RoboDK station: RDTSDemoBasketLineAndAGV.rdk

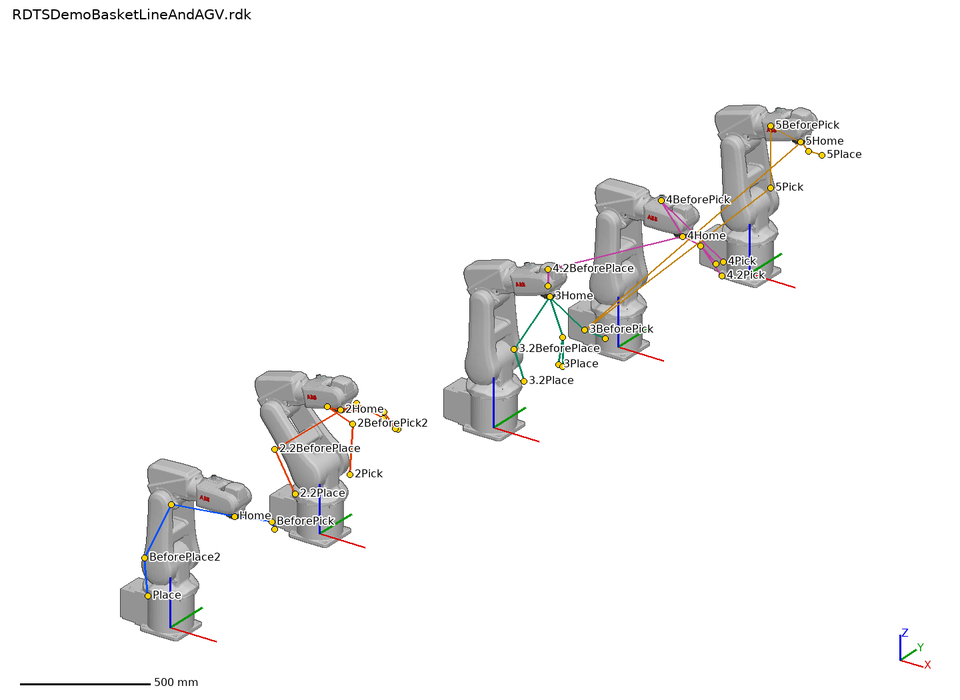
[picture v0: the station drawn from its stored meshes, robots at their saved joint values, targets as dots, program paths as lines]
Station RDTSDemoBasketLine (saved by RoboDK 5.6.0). Poses are relative to the parent item; angles as X-Y-Z fixed-axis rotations.
Station parameters (name, value as stored): 1MoveToPick, 0, 1MakePick, 0, 1PickObjOK, 0, 1MoveToPlace, 0, 1MakePlace, 0, 1PlaceObjOK, 1, 1Waitting, 1, 2MoveToPick, 0, 2MakePick, 0, 2PickObjOK, 0, 2MoveToPlace, 0, 2MakePlace, 0, 2PlaceObjOK, 0, 2Waitting, 1, 3MoveToPick, 0, 3MakePick, 0, 3PickObjOK, 0, 3MoveToPlace, 0, 3MakePlace, 0, 3PlaceObjOK, 0, 3Waitting, 1, 4MoveToPick, 0, 4MakePick, 0, 4PickObjOK, 0, 4MoveToPlace, 0, 4MakePlace, 0, 4PlaceObjOK, 0, 4Waitting, 1, 5MoveToPick, 0, 5MakePick, 0, 5PickObjOK, 0, 5MoveToPlace, 0, 5MakePlace, 0, 5PlaceObjOK, 0, 5Waitting, 1
  - frame Robot1Base at (0, 0, 0) mm
    - robot Robot1 (model ABB IRB 120-3/0.6): 6 axes, payload 3 kg, reach 580 mm, repeatability 0.01 mm, weight 25 kg
        modified DH rows (alpha deg, a mm, theta deg, d mm): 0, 0, 0, 290; -90, 0, -90, 0; 0, 270, 0, 0; -90, 70, 0, 302; 90, 0, 0, 0; -90, 0, 180, 72
        joint limits [-165, -110, -90, -160, -120, -400] to [165, 110, 70, 160, 120, 400]; home [0, 0, 0, 0, 0, 0]; saved at [0, 0, 0, 0, 90, 0]
    - target Home (Cartesian target) at (302, 0, 558) mm, rotated rx 180 ry 0 rz -180 deg; joints [0, 0, 0, 0, 90, 0] of Robot1
    - target BeforePick (Cartesian target) at (403.62, 104.76, 521.84) mm, rotated rx 179.56 ry -0.69 rz -179.99 deg; joints [14.447, 24.813, -22.689, 0.602, 88.437, 14.424] of Robot1
    - target Pick (Cartesian target) at (413.42, 104.99, 492) mm, rotated rx 179.56 ry -0.69 rz -179.99 deg; joints [14.149, 26.117, -18.91, 0.603, 83.358, 14.073] of Robot1
    - target AfterPick (Cartesian target) at (403.62, 104.76, 521.84) mm, rotated rx 179.56 ry -0.69 rz -179.99 deg; joints [14.447, 24.813, -22.689, 0.602, 88.437, 14.424] of Robot1
    - target BeforePlace (Cartesian target) at (41.23, -52.32, 557.95) mm, rotated rx -179.99 ry 0.01 rz 90.63 deg; joints [-51.75, -47.75, 30.07, -0.01, 107.68, 37.62] of Robot1
    - target BeforePlace2 (Cartesian target) at (26.38, -212.17, 388.44) mm, rotated rx 180 ry 0.01 rz 90.63 deg; joints [-82.912, -18.126, 47.312, -0.001, 60.804, 6.459] of Robot1
    - target Place (Cartesian target) at (41.74, -212.03, 229.97) mm, rotated rx -180 ry 0.01 rz 90.63 deg; joints [-78.863, 8.497, 59.917, -0.005, 21.575, 10.511] of Robot1
    - target AfterPlace (Cartesian target) at (26.38, -212.17, 388.44) mm, rotated rx 180 ry 0.01 rz 90.63 deg; joints [-82.912, -18.126, 47.312, -0.001, 60.804, 6.459] of Robot1
    - target AfterPlace2 (Cartesian target) at (41.23, -52.32, 557.95) mm, rotated rx -179.99 ry 0.01 rz 90.63 deg; joints [-51.75, -47.75, 30.07, -0.01, 107.68, 37.62] of Robot1
  - program RobotProg1 (31 instructions, listed below)
  - frame Robot2Base at (0, 1000, 0) mm
    - robot Robot2 (model ABB IRB 120-3/0.6): 6 axes, payload 3 kg, reach 580 mm, repeatability 0.01 mm, weight 25 kg
        modified DH rows (alpha deg, a mm, theta deg, d mm): 0, 0, 0, 290; -90, 0, -90, 0; 0, 270, 0, 0; -90, 70, 0, 302; 90, 0, 0, 0; -90, 0, 180, 72
        joint limits [-165, -110, -90, -160, -120, -400] to [165, 110, 70, 160, 120, 400]; home [0, 0, 0, 0, 0, 0]; saved at [0, -40.936, 28.088, 0, 105.49, 0]
    - target 2Home (Cartesian target) at (98.64, 0, 557.45) mm, rotated rx 180 ry -2.64 rz 180 deg; joints [0, -40.936, 28.088, 0, 105.49, 0] of Robot2
    - target 2BeforePick (Cartesian target) at (1.46, 49.24, 523.75) mm, rotated rx -179.78 ry 0.01 rz -91.44 deg; joints [88.62, -55.08, 38.94, -0.23, 106.13, 0] of Robot2
    - target 2BeforePick2 (Cartesian target) at (6.13, 213.1, 386.02) mm, rotated rx -179.78 ry 0 rz -89.11 deg; joints [88.428, -18.104, 47.764, -0.254, 60.33, -2.333] of Robot2
    - target 2Pick (Cartesian target) at (7.29, 189.51, 178.81) mm, rotated rx -179.78 ry 0 rz -89.11 deg; joints [87.881, 19.532, 64.824, -2.249, 5.635, -0.768] of Robot2
    - target 2AfterPick (Cartesian target) at (6.13, 213.1, 386.02) mm, rotated rx -179.78 ry 0 rz -89.11 deg; joints [88.428, -18.104, 47.764, -0.254, 60.33, -2.333] of Robot2
    - target 2AfterPick2 (Cartesian target) at (1.46, 49.24, 523.75) mm, rotated rx -179.78 ry 0.01 rz -91.44 deg; joints [88.62, -55.08, 38.94, -0.23, 106.13, 0] of Robot2
    - target 2BeforePlace (Cartesian target) at (113.67, 83.97, 556.76) mm, rotated rx -180 ry -2.64 rz -180 deg; joints [35.67, -32.578, 24.615, 1.564, 100.106, 35.915] of Robot2
    - target 2BeforePlace2 (Cartesian target) at (234.07, 92.8, 521.73) mm, rotated rx -180 ry -2.64 rz -180 deg; joints [21.351, -11.251, 17.104, 0.963, 86.608, 21.273] of Robot2
    - target 2Place (Cartesian target) at (300.85, 92.8, 493.46) mm, rotated rx -180 ry -2.64 rz -180 deg; joints [16.966, 1.709, 10.324, 0.781, 80.494, 16.82] of Robot2
    - target 2AfterPlace (Cartesian target) at (234.07, 92.8, 521.73) mm, rotated rx -180 ry -2.64 rz -180 deg; joints [21.351, -11.251, 17.104, 0.963, 86.608, 21.273] of Robot2
    - target 2AfterPlace2 (Cartesian target) at (113.67, 83.97, 556.76) mm, rotated rx -180 ry -2.64 rz -180 deg; joints [35.67, -32.578, 24.615, 1.564, 100.106, 35.915] of Robot2
    - target 2.2BeforePick (Cartesian target) at (235.43, 92.8, 551.14) mm, rotated rx -180 ry -2.64 rz -180 deg; joints [21.24, -9.919, 10.469, 0.957, 91.912, 21.252] of Robot2
    - target 2.2Pick (Cartesian target) at (290.1, 92.8, 493.96) mm, rotated rx 180 ry -2.64 rz -180 deg; joints [17.55, -0.469, 12.431, 0.807, 80.558, 17.4] of Robot2
    - target 2.2AfterPick (Cartesian target) at (235.43, 92.8, 551.14) mm, rotated rx -180 ry -2.64 rz -180 deg; joints [21.24, -9.919, 10.469, 0.957, 91.912, 21.252] of Robot2
    - target 2.2BeforePlace (Cartesian target) at (0, -302, 481.65) mm, rotated rx 180 ry 0 rz 90 deg; joints [-90, -1.686, 15.888, 0, 75.798, 0] of Robot2
    - target 2.2Place (Cartesian target) at (40.05, -221.68, 270.88) mm, rotated rx 180 ry 0 rz 90 deg; joints [-79.758, 0.841, 56.658, 0, 32.501, 10.242] of Robot2
    - target 2.2AfterPlace (Cartesian target) at (0, -302, 481.65) mm, rotated rx 180 ry 0 rz 90 deg; joints [-90, -1.686, 15.888, 0, 75.798, 0] of Robot2
  - program RobotProg2 (59 instructions, listed below)
  - frame Robot3Base at (11.58, 2148.25, 0) mm
    - robot Robot3 (model ABB IRB 120-3/0.6): 6 axes, payload 3 kg, reach 580 mm, repeatability 0.01 mm, weight 25 kg
        modified DH rows (alpha deg, a mm, theta deg, d mm): 0, 0, 0, 290; -90, 0, -90, 0; 0, 270, 0, 0; -90, 70, 0, 302; 90, 0, 0, 0; -90, 0, 180, 72
        joint limits [-165, -110, -90, -160, -120, -400] to [165, 110, 70, 160, 120, 400]; home [0, 0, 0, 0, 0, 0]; saved at [0, -2.008, -12.768, 0, 106.098, 0]
    - target 3Home (Cartesian target) at (263.04, 0, 632.56) mm, rotated rx 180 ry -1.32 rz -180 deg; joints [0, -2.008, -12.768, 0, 106.098, 0] of Robot3
    - target 3BeforePick (Cartesian target) at (354.26, 102.57, 474.34) mm, rotated rx -179.62 ry 0.29 rz -90.13 deg; joints [16.114, 12.475, 1.922, 0.178, 75.155, -73.797] of Robot3
    - target 3Pick (Cartesian target) at (363.26, 230.79, 389.57) mm, rotated rx -179.62 ry 0.29 rz -90.13 deg; joints [32.423, 28.064, -2.593, 0.044, 64.05, -57.463] of Robot3
    - target 3AfterPick (Cartesian target) at (354.26, 102.57, 474.34) mm, rotated rx -179.62 ry 0.29 rz -90.13 deg; joints [16.114, 12.475, 1.922, 0.178, 75.155, -73.797] of Robot3
    - target 3BeforePlace (Cartesian target) at (354.17, -42.25, 502) mm, rotated rx -179.54 ry 0.5 rz -180 deg; joints [-6.721, 9.918, -0.202, -0.408, 79.734, -6.652] of Robot3
    - target 3Place (Cartesian target) at (334.7, -43.23, 380.01) mm, rotated rx -179.54 ry 0.5 rz -180 deg; joints [-7.275, 9.557, 23.144, -0.474, 56.746, -7.02] of Robot3
    - target 3AfterPlace (Cartesian target) at (354.17, -42.25, 502) mm, rotated rx -179.54 ry 0.5 rz -180 deg; joints [-6.721, 9.918, -0.202, -0.408, 79.734, -6.652] of Robot3
    - target 3.2BeforePick (Cartesian target) at (354.17, -42.25, 502) mm, rotated rx -179.54 ry 0.5 rz -180 deg; joints [-6.721, 9.918, -0.202, -0.408, 79.734, -6.652] of Robot3
    - target 3.2Pick (Cartesian target) at (355.26, -44.09, 376.5) mm, rotated rx -179.54 ry 0.5 rz -180 deg; joints [-6.995, 13.95, 18.612, -0.476, 56.887, -6.738] of Robot3
    - target 3.2AfterPick (Cartesian target) at (354.17, -42.25, 502) mm, rotated rx -179.54 ry 0.5 rz -180 deg; joints [-6.721, 9.918, -0.202, -0.408, 79.734, -6.652] of Robot3
    - target 3.2BeforePlace (Cartesian target) at (302, -294.64, 535.14) mm, rotated rx 180 ry 0 rz -180 deg; joints [-44.294, 26.712, -27.845, 0, 91.133, -44.294] of Robot3
    - target 3.2Place (Cartesian target) at (347.56, -292.05, 411.65) mm, rotated rx 180 ry 0 rz -180 deg; joints [-40.04, 32.683, -13.41, 0, 70.727, -40.04] of Robot3
    - target 3.2AfterPlace (Cartesian target) at (302, -294.64, 535.14) mm, rotated rx -180 ry 0 rz 180 deg; joints [-44.294, 26.712, -27.845, 0, 91.133, -44.294] of Robot3
  - program RobotProg3 (55 instructions, listed below)
  - frame Robot4Base at (0, 3000, 0) mm
    - robot Robot4 (model ABB IRB 120-3/0.6): 6 axes, payload 3 kg, reach 580 mm, repeatability 0.01 mm, weight 25 kg
        modified DH rows (alpha deg, a mm, theta deg, d mm): 0, 0, 0, 290; -90, 0, -90, 0; 0, 270, 0, 0; -90, 70, 0, 302; 90, 0, 0, 0; -90, 0, 180, 72
        joint limits [-165, -110, -90, -160, -120, -400] to [165, 110, 70, 160, 120, 400]; home [0, 0, 0, 0, 0, 0]; saved at [0, 0, 0, 0, 90, 0]
    - target 4Home (Cartesian target) at (302, 0, 558) mm, rotated rx 180 ry 0 rz -180 deg; joints [0, 0, 0, 0, 90, 0] of Robot4
    - target 4BeforePick (Cartesian target) at (55.44, 208.73, 558) mm, rotated rx 180 ry 0 rz -90 deg; joints [75.125, -17.843, 15.366, 0, 92.477, -14.875] of Robot4
    - target 4Pick (Cartesian target) at (252.55, 343.75, 297.32) mm, rotated rx 180 ry 0 rz -98.96 deg; joints [53.695, 34.248, 6.452, 0, 49.299, -27.345] of Robot4
    - target 4AfterPick (Cartesian target) at (55.44, 208.73, 558) mm, rotated rx 180 ry 0 rz -90 deg; joints [75.125, -17.843, 15.366, 0, 92.477, -14.875] of Robot4
    - target 4BeforePlace (Cartesian target) at (400.62, -18.49, 552.3) mm, rotated rx 180 ry 0 rz -179.65 deg; joints [-2.642, 22.385, -25.18, 0, 92.795, -2.992] of Robot4
    - target 4Place (Cartesian target) at (479.11, -29.28, 501.07) mm, rotated rx 180 ry 0 rz -178.86 deg; joints [-3.497, 42.188, -44.67, 0, 92.482, -4.634] of Robot4
    - target 4AfterPlace (Cartesian target) at (400.62, -18.49, 552.3) mm, rotated rx 180 ry 0 rz -179.65 deg; joints [-2.642, 22.385, -25.18, 0, 92.795, -2.992] of Robot4
    - target 4.2BeforePick (Cartesian target) at (400.62, -18.49, 552.3) mm, rotated rx 180 ry 0 rz -179.65 deg; joints [-2.642, 22.385, -25.18, 0, 92.795, -2.992] of Robot4
    - target 4.2Pick (Cartesian target) at (500.88, -21.69, 451.45) mm, rotated rx 180 ry 0 rz -179.65 deg; joints [-2.48, 46.195, -41.782, 0, 85.586, -2.83] of Robot4
    - target 4.2AfterPick (Cartesian target) at (400.62, -18.49, 552.3) mm, rotated rx 180 ry 0 rz -179.65 deg; joints [-2.642, 22.385, -25.18, 0, 92.795, -2.992] of Robot4
    - target 4.2BeforePlace (Cartesian target) at (-46.76, -402.38, 479.67) mm, rotated rx 180 ry 0 rz 89.48 deg; joints [-96.629, 20.65, -9.266, 0, 78.616, -6.109] of Robot4
    - target 4.2Place (Cartesian target) at (-46.76, -402.38, 408.42) mm, rotated rx 180 ry 0 rz 89.48 deg; joints [-96.629, 21.955, 2.254, 0, 65.791, -6.109] of Robot4
    - target 4.2AfterPlace (Cartesian target) at (-46.76, -402.38, 479.67) mm, rotated rx 180 ry 0 rz 89.48 deg; joints [-96.629, 20.65, -9.266, 0, 78.616, -6.109] of Robot4
  - program RobotProg4 (55 instructions, listed below)
  - frame Robot5Base at (45.12, 3815.29, 0) mm
    - robot Robot5 (model ABB IRB 120-3/0.6): 6 axes, payload 3 kg, reach 580 mm, repeatability 0.01 mm, weight 25 kg
        modified DH rows (alpha deg, a mm, theta deg, d mm): 0, 0, 0, 290; -90, 0, -90, 0; 0, 270, 0, 0; -90, 70, 0, 302; 90, 0, 0, 0; -90, 0, 180, 72
        joint limits [-165, -110, -90, -160, -120, -400] to [165, 110, 70, 160, 120, 400]; home [0, 0, 0, 0, 0, 0]; saved at [0, -6.967, -7.658, 0, 105.716, 0]
    - target 5Home (Cartesian target) at (240.42, 0, 630) mm, rotated rx 180 ry -1.09 rz -180 deg; joints [0, -6.967, -7.658, 0, 105.716, 0] of Robot5
    - target 5BeforePick (Cartesian target) at (-65.99, 235.86, 518.13) mm, rotated rx -180 ry 0 rz -90 deg; joints [105.63, -13.451, 19.546, 0, 83.904, 15.63] of Robot5
    - target 5Pick (Cartesian target) at (-65.99, 235.86, 254.8) mm, rotated rx -180 ry 0 rz -90 deg; joints [105.63, 8.024, 53.076, 0, 28.9, 15.63] of Robot5
    - target 5AfterPick (Cartesian target) at (-65.99, 235.86, 518.13) mm, rotated rx -180 ry 0 rz -90 deg; joints [105.63, -13.451, 19.546, 0, 83.904, 15.63] of Robot5
    - target 5BeforePlace (Cartesian target) at (302.82, -36.16, 623.63) mm, rotated rx -180 ry -0.4 rz -180 deg; joints [-6.799, 5.822, -19.002, -0.048, 103.574, -6.81] of Robot5
    - target 5Place (Cartesian target) at (363.64, -36.16, 623.21) mm, rotated rx -180 ry -0.4 rz -180 deg; joints [-5.672, 20.893, -37.408, -0.041, 106.909, -5.683] of Robot5
    - target 5AfterPlace (Cartesian target) at (302.82, -36.16, 623.63) mm, rotated rx -180 ry -0.4 rz -180 deg; joints [-6.799, 5.822, -19.002, -0.048, 103.574, -6.81] of Robot5
  - program RobotProg5 (29 instructions, listed below)
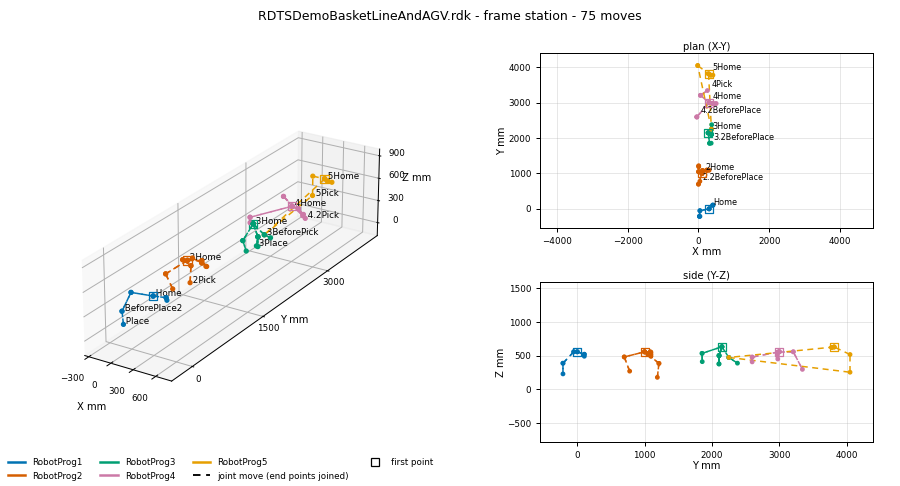
[picture p0: tool path of RDTSDemoBasketLineAndAGV.rdk in frame station, 75 of 75 moves have a stored position in this frame; points joined in program order, loops and branches not executed]

--- program RobotProg1 (robot Robot1) ---
  设置参考: Robot1Base
  MoveJ (Home)
  Set 1MakePick=0
  Set 1PickObjOK=0
  Set 1MakePlace=0
  Set 1PlaceObjOK=0
  Wait 1MoveToPick=1
  Set 1Waitting=0
  MoveJ (BeforePick)
  MoveJ (Pick)
  Set 1MakePick=1
  Wait 1PickObjOK=1
  Set 1MakePick=0
  暂停 2.0 s
  MoveJ (AfterPick)
  MoveJ (Home)
  Set 1Waitting=1
  Wait 1MoveToPlace=1
  Set 1Waitting=0
  MoveJ (BeforePlace)
  MoveJ (BeforePlace2)
  MoveJ (Place)
  Set 1MakePlace=1
  暂停 500 ms
  Wait 1PlaceObjOK=1
  Set 1MakePlace=0
  暂停 1.0 s
  MoveJ (AfterPlace)
  MoveJ (AfterPlace2)
  MoveJ (Home)
  Set 1Waitting=1

--- program RobotProg2 (robot Robot2) ---
  设置参考: Robot2Base
  MoveJ (2Home)
  Set 2MakePick=0
  Set 2PickObjOK=0
  Set 2MakePlace=0
  Set 2PlaceObjOK=0
  Wait 2MoveToPick=1
  Set 2Waitting=0
  MoveJ (2BeforePick)
  MoveJ (2BeforePick2)
  MoveJ (2Pick)
  Set 2MakePick=1
  Wait 2PickObjOK=1
  Set 2MakePick=0
  暂停 2.0 s
  MoveJ (2AfterPick)
  MoveJ (2AfterPick2)
  MoveJ (2Home)
  Set 2Waitting=1
  Wait 2MoveToPlace=1
  Set 2Waitting=0
  MoveJ (2BeforePlace)
  MoveJ (2BeforePlace2)
  MoveJ (2Place)
  Set 2MakePlace=1
  Wait 2PlaceObjOK=1
  Set 2MakePlace=0
  暂停 1.0 s
  MoveJ (2AfterPlace)
  MoveJ (2AfterPlace2)
  MoveJ (2Home)
  Set 2Waitting=1
  暂停 2.5 s
  Set 2MakePick=0
  Set 2PickObjOK=0
  Set 2MakePlace=0
  Set 2PlaceObjOK=0
  Wait 2MoveToPick=1
  Set 2Waitting=0
  MoveJ (2.2BeforePick)
  MoveJ (2.2Pick)
  Set 2MakePick=1
  Wait 2PickObjOK=1
  Set 2MakePick=0
  暂停 2.0 s
  MoveJ (2.2AfterPick)
  MoveJ (2Home)
  Set 2Waitting=1
  Wait 2MoveToPlace=1
  Set 2Waitting=0
  MoveJ (2.2BeforePlace)
  MoveJ (2.2Place)
  Set 2MakePlace=1
  Wait 2PlaceObjOK=1
  Set 2MakePlace=0
  暂停 1.0 s
  MoveJ (2.2AfterPlace)
  MoveJ (2Home)
  Set 2Waitting=1

--- program RobotProg3 (robot Robot3) ---
  设置参考: Robot3Base
  MoveJ (3Home)
  Set 3MakePick=0
  Set 3PickObjOK=0
  Set 3MakePlace=0
  Set 3PlaceObjOK=0
  Wait 3MoveToPick=1
  Set 3Waitting=0
  MoveJ (3BeforePick)
  MoveJ (3Pick)
  Set 3MakePick=1
  Wait 3PickObjOK=1
  Set 3MakePick=0
  暂停 2.0 s
  MoveJ (3AfterPick)
  MoveJ (3Home)
  Set 3Waitting=1
  Wait 3MoveToPlace=1
  Set 3Waitting=0
  MoveJ (3BeforePlace)
  MoveJ (3Place)
  Set 3MakePlace=1
  Wait 3PlaceObjOK=1
  Set 3MakePlace=0
  暂停 1.0 s
  MoveJ (3AfterPlace)
  MoveJ (3Home)
  Set 3Waitting=1
  暂停 2.5 s
  Set 3MakePick=0
  Set 3PickObjOK=0
  Set 3MakePlace=0
  Set 3PlaceObjOK=0
  Wait 3MoveToPick=1
  Set 3Waitting=0
  MoveJ (3.2BeforePick)
  MoveJ (3.2Pick)
  Set 3MakePick=1
  Wait 3PickObjOK=1
  Set 3MakePick=0
  暂停 2.0 s
  MoveJ (3.2AfterPick)
  MoveJ (3Home)
  Set 3Waitting=1
  Wait 3MoveToPlace=1
  Set 3Waitting=0
  MoveJ (3.2BeforePlace)
  MoveJ (3.2Place)
  Set 3MakePlace=1
  Wait 3PlaceObjOK=1
  Set 3MakePlace=0
  暂停 1.0 s
  MoveJ (3.2AfterPlace)
  MoveJ (3Home)
  Set 3Waitting=1

--- program RobotProg4 (robot Robot4) ---
  设置参考: Robot4Base
  MoveJ (4Home)
  Set 4MakePick=0
  Set 4PickObjOK=0
  Set 4MakePlace=0
  Set 4PlaceObjOK=0
  Wait 4MoveToPick=1
  Set 4Waitting=0
  MoveJ (4BeforePick)
  MoveJ (4Pick)
  Set 4MakePick=1
  Wait 4PickObjOK=1
  Set 4MakePick=0
  暂停 2.0 s
  MoveJ (4AfterPick)
  MoveJ (4Home)
  Set 4Waitting=1
  Wait 4MoveToPlace=1
  Set 4Waitting=0
  MoveJ (4BeforePlace)
  MoveJ (4Place)
  Set 4MakePlace=1
  Wait 4PlaceObjOK=1
  Set 4MakePlace=0
  暂停 1.0 s
  MoveJ (4AfterPlace)
  MoveJ (4Home)
  Set 4Waitting=1
  暂停 2.5 s
  Set 4MakePick=0
  Set 4PickObjOK=0
  Set 4MakePlace=0
  Set 4PlaceObjOK=0
  Wait 4MoveToPick=1
  Set 4Waitting=0
  MoveJ (4.2BeforePick)
  MoveJ (4.2Pick)
  Set 4MakePick=1
  Wait 4PickObjOK=1
  Set 4MakePick=0
  暂停 2.0 s
  MoveJ (4.2AfterPick)
  MoveJ (4Home)
  Set 4Waitting=1
  Wait 4MoveToPlace=1
  Set 4Waitting=0
  MoveJ (4.2BeforePlace)
  MoveJ (4.2Place)
  Set 4MakePlace=1
  Wait 4PlaceObjOK=1
  Set 4MakePlace=0
  暂停 1.0 s
  MoveJ (4.2AfterPlace)
  MoveJ (4Home)
  Set 4Waitting=1

--- program RobotProg5 (robot Robot5) ---
  设置参考: Robot5Base
  MoveJ (5Home)
  Set 5MakePick=0
  Set 5PickObjOK=0
  Set 5MakePlace=0
  Set 5PlaceObjOK=0
  Wait 5MoveToPick=1
  Set 5Waitting=0
  MoveJ (5BeforePick) -> target 3BeforePick
  MoveJ (5Pick)
  Set 5MakePick=1
  Wait 5PickObjOK=1
  Set 5MakePick=0
  暂停 2.0 s
  MoveJ (5AfterPick)
  MoveJ (5Home)
  Set 5Waitting=1
  Wait 5MoveToPlace=1
  Set 5Waitting=0
  MoveJ (5BeforePlace)
  MoveJ (5Place)
  Set 5MakePlace=1
  暂停 500 ms
  Wait 5PlaceObjOK=1
  Set 5MakePlace=0
  暂停 1.0 s
  MoveJ (5AfterPlace)
  MoveJ (5Home)
  Set 5Waitting=1
